short summary
=================
Tests timeout behavior of the cycle manager.
Verifies timeout configuration and automatic transition to timeout step.

.. <legal notes>

legal notes
=================
| SPDX-FileCopyrightText: © 2025 ekvip automation GmbH <info@ekvip.de>
| SPDX-License-Identifier: Apache-2.0
| For details check: Apache-2.0_

.. _Apache-2.0: https://www.apache.org/licenses/LICENSE-2.0

.. </legal notes>

*)
METHOD PRIVATE testTimeoutBehavior
VAR_INST
	testState : INT;
	timeoutTimer : TON;
END_VAR
RETURN( THIS^.testSuiteAborted OR_ELSE  NOT TcUnit.TEST_ORDERED(THIS^.getTestNameFor('testTimeoutBehavior')));

CASE testState OF
0: // Initialize
	THIS^.resetCycleManager();
	iConfiguration := cycleManager;
	iCycleManager := cycleManager;
	testState := 10;
	
10: // Configure timeout
	cycleManager.update(execute := TRUE);
	
	// Set sequence timeout
	iConfiguration.configuration.sequence.timeout := T#100MS;
	iConfiguration.configuration.sequence.timeoutStep := 999;
	
	iCycleManager.proceedWith(10);
	testState := 20;
	
20: // Wait for timeout
	cycleManager.update(execute := TRUE); // Disable step control to trigger timeout
	// Start timer to track timeout
	timeoutTimer(IN := cycleManager.executeStep, PT := T#110MS);
	CASE cycleManager.step.current OF 
	10:
		IF timeoutTimer.Q THEN
			AssertTrue(
				Condition := FALSE,
				Message := 'Cyclemanager timeout not triggered in time'
			);
			testState := 100;
		END_IF
	999:
		testState := 30;
	ELSE
		AssertTrue(
			Condition := FALSE,
			Message := 'wrong step after timeout monitoring detected'
		);
		testState := 100;
	END_CASE
	
30:
	AssertTrue(
		Condition := cycleManager.errors.isInErrorStep,
		Message := 'Timeout step should be marked as error step'
	);
	cycleManager.proceedWith(10);
	testState := 40;
40:
	cycleManager.update(execute := TRUE);
	cycleManager.configuration.step.timeoutStep := 666;
	cycleManager.configuration.step.timeout := T#50MS;
	timeoutTimer(IN := cycleManager.executeStep, PT := T#60MS);
	CASE cycleManager.step.current OF
	10:
		IF timeoutTimer.Q THEN
			AssertTrue(
				Condition := FALSE,
				Message := 'Cyclemanager timeout not triggered in time'
			);
			testState := 100;
		END_IF
	666:
		testState := 50;
		AssertTrue(
			Condition := cycleManager.errors.isInErrorStep,
			Message := 'Timeout step should be marked as error step'
		);
		cycleManager.proceedWith(10);	
	999:
		AssertTrue(
			Condition := FALSE,
			Message := 'global sequence timeout triggered instead of local step configuration'
		);
		testState := 100;
	ELSE
		AssertTrue(
			Condition := FALSE,
			Message := 'wrong step after timeout monitoring detected'
		);
		testState := 100;	
	END_CASE
50:
	// Wait for timeout
	cycleManager.update(execute := TRUE); // Disable step control to trigger timeout
	// Start timer to track timeout
	timeoutTimer(IN := cycleManager.executeStep, PT := T#110MS);
	CASE cycleManager.step.current OF 
	10:
		IF timeoutTimer.Q THEN
			AssertTrue(
				Condition := FALSE,
				Message := 'Cyclemanager timeout not triggered in time'
			);
			testState := 100;
		END_IF
	999:
		testState := 100;
	ELSE
		AssertTrue(
			Condition := FALSE,
			Message := 'wrong step after timeout monitoring detected'
		);
		testState := 100;
	END_CASE
100:
	TEST_FINISHED();
END_CASE
END_METHOD

(*

short summary
=================
Tests the waitFor() method behavior.
Verifies that the cycle manager waits for a boolean condition before proceeding.

.. <legal notes>

legal notes
=================
| SPDX-FileCopyrightText: © 2025 ekvip automation GmbH <info@ekvip.de>
| SPDX-License-Identifier: Apache-2.0
| For details check: Apache-2.0_

.. _Apache-2.0: https://www.apache.org/licenses/LICENSE-2.0

.. </legal notes>

*)
METHOD PRIVATE testWaitForMethod
VAR_INST
	testState : INT;
	waitCondition : BOOL;
	cycleCount : INT;
END_VAR
VAR
	foo :POINTER TO BYTE := ADR(waitCondition);
	bar : ARRAY [0..1] OF DINT := [10, 11];
	
END_VAR
RETURN( THIS^.testSuiteAborted OR_ELSE  NOT TcUnit.TEST_ORDERED(THIS^.getTestNameFor('testWaitForMethod')));

CASE testState OF
0: // Initialize
	THIS^.resetCycleManager();
	iCycleManager := cycleManager;
	waitCondition := FALSE;
	cycleCount := 0;
	testState := 10;
	
10: // Start and move to test step
	cycleManager.update(execute := TRUE);
	iCycleManager.proceedWith(10);
	testState := 20;
	cycleManager.update(execute := TRUE);
	
20: // Test waitFor
	// After 3 cycles, set condition true
	cycleCount := cycleCount + 1;
	IF cycleCount >= 4 THEN
		waitCondition := TRUE;
		testState := 30;
		cycleCount := 0;
	END_IF
	iCycleManager.waitFor(value := waitCondition);
	
	cycleManager.update(execute := TRUE);
	// Wait should keep step busy
	AssertEquals_DINT(
		Expected := bar[foo^],
		Actual := iCycleManager.step.current,
		Message := 'Step should only change when waitForCondition is true'
	);
	waitCondition := FALSE;
	
30: // Verify proceeded to next step
	cycleManager.update(execute := TRUE);
	cycleManager.waitFor(TRUE);
	AssertEquals_DINT(
		Expected := 11, // Default step width is 1
		Actual := iCycleManager.step.current,
		Message := 'Should not proceed without update call'
	);
	cycleManager.update(execute := TRUE);
	AssertEquals_DINT(
		Expected := 12, // Default step width is 1
		Actual := iCycleManager.step.current,
		Message := 'Should proceed after update call'
	);
	
	TEST_FINISHED();	
END_CASE
END_METHOD

END_FUNCTION_BLOCK

(* stored: Version 1.1.0.1
   POU InterfaceTests: Id {3bea2955-06fa-4ed1-baaa-d2be70c1833d}, SpecialFunc None
   Folder internal: Id {1480186d-90a3-4194-b6c9-d81544f9a9b9}
   Method abortTestsuite: Id {e3775ff2-ae77-4610-9d91-9f08d63aa5ee}
   Method FB_init: Id {37f4df8a-d3cf-4fc0-8df8-3135f90255b2}
   Method getTestNameFor: Id {12345678-90ab-cdef-1234-567890abcdef}
   Method resetCycleManager: Id {8b34567c-def0-1234-5678-901234567890}
   Method testBasicStepNavigation: Id {a1b2c3d4-e5f6-7890-abcd-ef1234567890}
   Method testEnterMethod: Id {b2c3d4e5-f6a7-8901-bcde-f23456789012}
   Method testErrorAcknowledgeMethod: Id {74956b43-0611-4c90-8a90-ca45cc66f60a}
   Method testErrorHandleMethod: Id {b8901234-5678-90ab-cdef-901234567890}
   Method testErrorStepConfig: Id {23b0dca8-3dd9-4282-b3aa-d5cc6ee2ece5}
   Method testEvaluateMethod: Id {e5f6a7b8-9012-3456-efab-678901234567}
   Method testExecuteCommandMethod: Id {d4e5f6a7-b890-1234-defa-567890123456}
   Method testExecuteStepProperty: Id {5a123456-7890-bcde-2345-678901234567}
   Method testFluentInterfaceChaining: Id {25678901-cdef-1234-5678-890123456121}
   Method testInterfaceNullSafety: Id {36789012-bcde-0123-4567-890123456232}
   Method testLeaveMethod: Id {c3d4e5f6-a7b8-9012-cdef-345678901234}
   Method testMultipleStepConfigurations: Id {45de67fa-89bc-0123-defa-456789012345}
   Method testPauseErrorIntegration: Id {789abcde-f012-3456-7890-abcdef012345}
   Method testPauseResumeBehavior: Id {03456789-abcd-f012-3456-6789012340ef}
   Method testProceedMethods: Id {a7b89012-3456-789a-bcde-890123456789}
   Method testStateProperty: Id {e1234567-89ab-def0-1234-456789012cde}
   Method testStepConfigurationReset: Id {56ef78ab-90cd-1234-efab-567890123456}
   Method testStepPauseOverride: Id {12ab34cd-56ef-7890-abcd-ef1234567890}
   Method testSteppingWithStepControl: Id {67fa89bc-def0-3456-7890-bcdef1234567}
   Method testStepProperties: Id {d0123456-789b-cdef-0123-345678901bcd}
   Method testStepSteppingOverride: Id {23bc45de-67fa-8901-bcde-f23456789012}
   Method testStepStopRequestOverride: Id {34cd56ef-78ab-9012-cdef-345678901234}
   Method testStepWidthConfig: Id {c9012345-678a-bcde-f012-234567890abc}
   Method testStopRequestModes: Id {14567890-bcde-0123-4567-789012345010}
   Method testSuccessRequiredConfig: Id {73513dd3-bfb8-44e4-91fd-b66a512db13c}
   Method testTimeoutBehavior: Id {f2345678-9abc-ef01-2345-567890123def}
   Method testWaitForMethod: Id {f6a7b890-1234-5678-fabc-789012345678} *)
